FUNCTION IsSome : BOOL
VAR_INPUT
	eResult			: Result;
END_VAR
VAR_OUTPUT
	eCarry			: Result;
END_VAR

IsSome := eResult <> 0;
eCarry := eResult;

END_FUNCTION

(* stored: Version 1.1.0.1
   POU IsSome: Id {a98731ff-27dc-440b-b01b-ce65cfe43b72}, SpecialFunc None *)
